// TIA Portal V16 export
// export: Created 2024-09-05T17:39:24.9034378Z, ExportSetting WithDefaults, DisplayName Totally Integrated Automation Portal, DisplayVersion V16 Update 6, DisplayName TIA Portal Version Control Interface, DisplayVersion V16 Update 2, DisplayName TIA Portal Openness, DisplayVersion V16 Update 6, DisplayName STEP 7 Professional, DisplayVersion V16 Update 6, DisplayName STEP 7 Safety, DisplayVersion V16, DisplayName WinCC Advanced, DisplayVersion V16 Update 6
DATA_BLOCK "5. Call_M005_VARIABILITY_DB"   // DB2005
VERSION : 0.1
// stored: AutoNumber false, DBAccessibleFromOPCUA true, InstanceOfName 5. Call_M005_VARIABILITY, InstanceOfType FB
"5. Call_M005_VARIABILITY"
   // VAR_INPUT
   //    "type" : WString;
   //    businessGroup : WString;
   //    technoCode : WString;
   //    location : WString;
   //    defectTypeCode : WString;
   //    defectNumber : Array[1..32] of DInt;
   //    x : Bool;
   // END_VAR
   // VAR_OUTPUT
   //    variabilityCode : WString[8];
   //    status : WString;
   // END_VAR
   // VAR
   //    variabilityIndex : Array[1..32] of WString[1];
   //    actualValue : Array[1..32] of DInt;
   //    timestamp : DTL;
   //    datestring : String;
   //    aux : Struct
   //       "bool" : Bool;
   //       idx : Int;
   //       "dword" : DWord;
   //       dword2 : DWord;
   //       tempArray : Array[1..32] of Bool;
   //       tempArray2 : Array[1..32] of Bool;
   //    END_STRUCT;
   // END_VAR
BEGIN
END_DATA_BLOCK
